{attribute addProperty BoxType "BK1120-0000-0020"}
{attribute addProperty Id "Term_380_KL1002KL1002_D229A9CA00"}
{attribute addProperty CRC "760044134"}
{attribute addProperty SizeInBites "0"}
{attribute addProperty SizeInBytes "0"}
TYPE A_0007_BK1120_0000_0020_2D4D5A66 EXTENDS BK1120_A5F67C82 :
STRUCT
	{attribute addProperty Name "Term_380_KL1002"}
	Term_380_KL1002 : KL1002_D229A9CA;
END_STRUCT
END_TYPE

(* stored: Version 1.2.0.0, ProductVersion 3.1.4024.9
   DUT A_0007_BK1120_0000_0020_2D4D5A66: Id {0a3269e9-85c4-4bf1-b502-5c0ed25ba298} *)
